TYPE ST_Siemens_data_outputs :
STRUCT
	T01_outlet : BOOL;
	T02_outlet : BOOL;
	Outlet_pump_motor : BOOL;
	Conveyor_motor : BOOL;
	T01_inlet : BOOL;
	T02_inlet : BOOL;	
END_STRUCT
END_TYPE

(* stored: Version 1.1.0.1, ProductVersion 3.1.4024.11
   DUT ST_Siemens_data_outputs: Id {2bba3856-728b-43d8-9a3f-450df304984d} *)
